GLOBALCONSTANTS DefaultPool_TC-SC_Numeric (* Numeric object pool constants (ID, Scale, Offset, Decimals) *)
  PACKAGE Uebungen::const::UT::TC-SC;
END_GLOBALCONSTANTS
